(* PLC project SafeLOGIC, BrAutomation SafeDESIGNER  5.24.1.0 *)
(* stored: companyURL http://www.br-automation.com, creationDateTime Mon Dec 15 17:46:18 2025 *)

PROGRAM Main

(* FBD diagram, written out as Structured Text *)
(* Function 03/04 - Oil pressure min/maximum *)
(* Actual oil pressure [mbar] *)
xSCALE_F03_AI_Pr_EO(sX := sAI_Pr_EO, sX1 := SAFEDINT#4000, sX2 := SAFEDINT#20000, sY1 := SAFEDINT#0, sY2 := SAFEDINT#10000, sbSafeCurrentOK := sbSafeCurrentOK_AI_Pr_EO);
siPr_EO := xSCALE_F03_AI_Pr_EO.sY_Scal;
(* Alarm *)
(* Safety loop *)
bAMM_A2387 := xSCALE_F03_AI_Pr_EO.bAMM_MSF;
iOUT_F03_Pr_EO := xSCALE_F03_AI_Pr_EO.iOUT_Y_Scal;
(* Measurement signal OK *)
sbPr_EO_MsOK := xSCALE_F03_AI_Pr_EO.sbMsOK;
sbSL_OK_EO_Ms := xSCALE_F03_AI_Pr_EO.sbSL_OK;
(* Actual oil pressure after pump [mbar] *)
xSCALE_F04_AI_Pr_EOaP(sX := sAI_Pr_EOaP, sX1 := SAFEDINT#4000, sX2 := SAFEDINT#20000, sY1 := SAFEDINT#0, sY2 := SAFEDINT#16000, sbSafeCurrentOK := sbSafeCurrentOK_AI_Pr_EOaP);
siPr_EOaP := xSCALE_F04_AI_Pr_EOaP.sY_Scal;
(* Alarm *)
(* Safety loop *)
bAMM_A2393 := xSCALE_F04_AI_Pr_EOaP.bAMM_MSF;
iOUT_F04_Pr_EOaP := xSCALE_F04_AI_Pr_EOaP.iOUT_Y_Scal;
(* Measurement signal OK *)
sbPr_EOaP_MsOK := xSCALE_F04_AI_Pr_EOaP.sbMsOK;
sbSL_OK_EOaP_Ms := xSCALE_F04_AI_Pr_EOaP.sbSL_OK;
(* Check oil pumps *)
(* All oil pumps off for 2min *)
(* Elapsed time *)
xELAPSED_TIME_EO(IN := BOOL_TO_SAFEBOOL(bIN_EO_PumpsOff), PT := SAFETIME#120s);
sbEO_PumpsOff_120s := xELAPSED_TIME_EO.Q;
iOUT_F04_EO_PumpsOff_2m_ET := xELAPSED_TIME_EO.iOUT_ET;
(* Pressure Minimum *)
(* Alarm *)
xINTERPOLATION_F03_Pr_EO_Min(sX := siN_EngAct, sX1 := PARA_N_Pr_EO_LoLo_Lim1, sX2 := PARA_N_Pr_EO_LoLo_Lim2, sY1 := PARA_Pr_EO_LoLo_LimN1, sY2 := PARA_Pr_EO_LoLo_LimN2);
xKeepAMM_2s_A2386(sbAMMxxxx := OR_S(GE_S(siPr_EO, xINTERPOLATION_F03_Pr_EO_Min.sY_Out), LT_S(siN_EngAct, PARA_N_Pr_EO_LoLo_Lim1), NOT_S(sbPr_EO_MsOK)));
bAMM_A2386 := xKeepAMM_2s_A2386.bAMMxxxx;
(* Plausibility check *)
(* Oil pressure at standstill [mbar] *)
xSET_F03_Pr_EO_Standstill(sbStoreValue := AND_S(sbEO_PumpsOff_120s, sbN_Standstill, sbPr_EO_MsOK), siValue := siPr_EO);
siPr_EO_Standstill := xSET_F03_Pr_EO_Standstill.siValue_Stored;
iOUT_F03_Pr_EO_Standstill := SAFEDINT_TO_DINT(xSET_F03_Pr_EO_Standstill.siValue_Stored);
(* Alarm *)
xR_TRIG_F03_Nom90(CLK := sbN_EngAct_Nom90_10s);
xKeepAMM_2s_A2388(sbAMMxxxx := OR_S(NOT_S(sbPr_EO_MsOK), AND_S(OR_S(NOT_S(xR_TRIG_F03_Nom90.Q), GE_S(SUB_S(siPr_EO, siPr_EO_Standstill), PARA_Pr_EO_Diff_EngStop)), OR_S(LE_S(siPr_EO, PARA_Pr_EO_HiHi_EngStop), NOT_S(AND_S(sbEO_PumpsOff_120s, sbN_Standstill_60s))))));
bAMM_A2388 := xKeepAMM_2s_A2388.bAMMxxxx;
(* Maximum deviation to pressure sensor after pump *)
(* Pressure difference [mbar] *)
xDEV_EO(sInput_1 := siPr_EO, sInput_2 := siPr_EOaP);
iOUT_F03_Pr_EO_Diff := xDEV_EO.iOUT_Diff;
(* Pressure difference OK *)
sbPr_EO_DiffOK := xDEV_EO.sbDiffOK;
siPr_EO_Diff := xDEV_EO.sDiff;
bOUT_F03_Pr_EO_DiffOK := xDEV_EO.bOUT_DiffOK;
(* Alarm *)
xKeepAMM_2s_A2389(sbAMMxxxx := NOT_S(AND_S(OR_S(GT_S(siPr_EO_Diff, PARA_Pr_EO_HiHi_Diff), NOT_S(sbPr_EO_DiffOK)), sbN_Standstill, sbEO_PumpsOff_120s, sbPr_EO_MsOK, sbPr_EOaP_MsOK)));
bAMM_A2389 := xKeepAMM_2s_A2389.bAMMxxxx;
(* Pressure Maximum (Sensor drift) *)
(* Alarm *)
xTOF_F03_Pr_EO_HiHi(IN := LE_S(siPr_EO, PARA_Pr_EO_HiHi_Check), PT := SAFETIME#10s);
xKeepAMM_2s_A2390(sbAMMxxxx := OR_S(xTOF_F03_Pr_EO_HiHi.Q, NOT_S(sbPr_EO_MsOK)));
bAMM_A2390 := xKeepAMM_2s_A2390.bAMMxxxx;
(* Frozen sensor value *)
(* Alarm *)
(* Elapsed time *)
xFROZEN_EO(siPr := siPr_EO, siPr_saved := siPr_EO_Saved, sbGV_Closed := sbGasValves_Closed, sbN_Nom90_10s := sbN_EngAct_Nom90_10s);
iOUT_F03_Pr_EO_Fr_1m_ET := xFROZEN_EO.iOUT_Pr_Frozen_1m_ET;
bAMM_A2391 := xFROZEN_EO.bError_Frozen;
(* Save actual value *)
siPr_EO_Saved := siPr_EO;
(* Safety loop *)
(* Safety loop *)
sbF03_OK_Oil_Pr_Min := AND_S(BOOL_TO_SAFEBOOL(bAMM_A2386), sbSL_OK_EO_Ms, BOOL_TO_SAFEBOOL(bAMM_A2388), BOOL_TO_SAFEBOOL(bAMM_A2389), BOOL_TO_SAFEBOOL(bAMM_A2390), BOOL_TO_SAFEBOOL(bAMM_A2391));
(* HMI - Oil pressure min OK *)
(* Oil pressure MIN OK *)
bOUT_F03_OK := SAFEBOOL_TO_BOOL(AND_S(sbN_EngAct_Nom90_10s, sbGasValves_Open, sbF03_OK_Oil_Pr_Min));
(* Release signal after error *)
(* Reset channel error *)
sbSafeRelease_AI_Pr_EO := BOOL_TO_SAFEBOOL(bIN_Reset_sPLC);
(* Pressure Maximum *)
(* Alarm *)
xKeepAMM_2s_A2392(sbAMMxxxx := OR_S(LT_S(siPr_EOaP, PARA_Pr_EOaP_HiHi), NOT_S(sbPr_EOaP_MsOK)));
bAMM_A2392 := xKeepAMM_2s_A2392.bAMMxxxx;
(* Plausibility check *)
(* Oil pressure at standstill [mbar] *)
xSET_F04_Pr_EOaP_Standstill(sbStoreValue := AND_S(sbEO_PumpsOff_120s, sbN_Standstill, sbPr_EOaP_MsOK), siValue := siPr_EOaP);
siPr_EOaP_Standstill := xSET_F04_Pr_EOaP_Standstill.siValue_Stored;
iOUT_F04_Pr_EOaP_Standstill := SAFEDINT_TO_DINT(xSET_F04_Pr_EOaP_Standstill.siValue_Stored);
(* Alarm *)
xR_TRIG_F04_Nom90(CLK := sbN_EngAct_Nom90_10s);
xKeepAMM_2s_A2394(sbAMMxxxx := OR_S(NOT_S(sbPr_EOaP_MsOK), AND_S(OR_S(NOT_S(xR_TRIG_F04_Nom90.Q), GE_S(SUB_S(siPr_EOaP, siPr_EOaP_Standstill), PARA_Pr_EOaP_Diff_EngStop)), OR_S(LE_S(siPr_EOaP, PARA_Pr_EOaP_HiHi_EngStop), NOT_S(AND_S(sbEO_PumpsOff_120s, sbN_Standstill_60s))))));
bAMM_A2394 := xKeepAMM_2s_A2394.bAMMxxxx;
(* Frozen sensor value *)
(* Alarm *)
(* Elapsed time *)
xFROZEN_EOaP(siPr := siPr_EOaP, siPr_saved := siPr_EOaP_Saved, sbGV_Closed := sbGasValves_Closed, sbN_Nom90_10s := sbN_EngAct_Nom90_10s);
iOUT_F04_Pr_EOaP_Fr_1m_ET := xFROZEN_EOaP.iOUT_Pr_Frozen_1m_ET;
bAMM_A2395 := xFROZEN_EOaP.bError_Frozen;
(* Save actual value *)
siPr_EOaP_Saved := siPr_EOaP;
(* Safety loop *)
(* Safety loop *)
sbF04_OK_Oil_Pr_Max := AND_S(BOOL_TO_SAFEBOOL(bAMM_A2392), sbSL_OK_EOaP_Ms, BOOL_TO_SAFEBOOL(bAMM_A2394), BOOL_TO_SAFEBOOL(bAMM_A2395));
(* HMI - Oil pressure max OK *)
(* Oil pressure MAX OK *)
bOUT_F04_OK := SAFEBOOL_TO_BOOL(AND_S(sbN_EngAct_Nom90_10s, sbGasValves_Open, sbF04_OK_Oil_Pr_Max));
(* Release signal after error *)
(* Reset channel error *)
sbSafeRelease_AI_Pr_EOaP := BOOL_TO_SAFEBOOL(bIN_Reset_sPLC);
END_PROGRAM
